FUNCTION A_USINT : ST_Arg
VAR_INPUT
	nNumber	: REFERENCE TO USINT;
END_VAR

IF __ISVALIDREF(nNumber) THEN
	A_USINT.eType := E_ArgType.USIntArg;
	A_USINT.pData := ADR(nNumber);
	A_USINT.nSize := SIZEOF(USINT);
END_IF

END_FUNCTION

(* stored: Version 1.1.0.1, ProductVersion 3.1.4024.15
   POU A_USINT: Id {55d6fcb6-3a9f-4fd8-b1c8-2c77ebf51bca}, SpecialFunc None *)
